//==================================================================================================
//								RJM Maszyny sp. z o.o.
//									13.05.2022
//	Obsługa silonwika z zawrorem 5 na 2 - 1 cewka
//	Realizacja wysuwania i chowania tłoczyska dla jednej cewki zwrócenie pozycji skrajnych
// 	v1.0	|| TC v 3.1.4024.22		|| - pierwsza wersja
//==================================================================================================
FUNCTION_BLOCK FB_Silownik_5na2_1Cewka EXTENDS FB_SIlownikBaza
VAR_INPUT
END_VAR
VAR_OUTPUT
END_VAR
VAR
END_VAR

METHOD Praca : BOOL
VAR_INPUT
END_VAR
SUPER^.Praca ();

IF (bPrzesuwanieWStroneKonca AND NOT bCewkaA) THEN
	bCewkaA									:= TRUE;
END_IF
IF  (bPrzesuwanieWStronePoczatku AND bCewkaA) THEN
	bCewkaA									:= FALSE;
END_IF
END_METHOD

END_FUNCTION_BLOCK

(* stored: Version 1.1.0.1, ProductVersion 3.1.4024.11
   POU FB_Silownik_5na2_1Cewka: Id {7381a165-2b77-46aa-97cc-7d9eb8e66228}, SpecialFunc None
   Method Praca: Id {c55b7c92-6fd0-4798-927c-ea98c74822a1} *)
